(* IEC 61131-3 sources: Industry-PLC-LLM/data/PLCBEAD_repo/PLCBEAD_PLCEmbed-main/PLC-BEAD/Source/GEB/MUL_ADD, 1 file *)

(* ---- MUL_ADD.ST ---- *)
FUNCTION MUL_ADD:REAL

	VAR_INPUT
		X :	REAL;
		K :	REAL;
		O :	REAL;
	END_VAR

	MUL_ADD := X * K + O;

END_FUNCTION

PROGRAM program0
	VAR
		X :	REAL;
		K :	REAL;
		O :	REAL;

		OUT : REAL;
	END_VAR

	OUT := MUL_ADD(X, K, O);

END_PROGRAM
